FUNCTION_BLOCK FB_WatsAppResponse
VAR_INPUT
	bSend             : BOOL;
END_VAR
VAR_OUTPUT
	wind_speed		  : Lreal;
	bBusy             : BOOL;
    bError            : BOOL;
END_VAR
VAR
	fbRequest         : FB_IotHttpRequest;
    fbJson            : FB_JsonDomParser;
    nState            : UDINT;
    RisingEdge        : R_TRIG;

    bGetContentResult : BOOL;
    sContent          : STRING(511);

    bGetJsonResult    : BOOL;
    jsonDoc           : SJsonValue;
    jsonVal           : SJsonValue;
	jsonWind           : SJsonValue;

    nReqCount         : UDINT;
    nResCount         : UDINT;
    nValidResCount    : UDINT;
    nErrCount         : UDINT;
	bHasMember		  : BOOL;
	bHasMember2		  : BOOL;
END_VAR
VAR_IN_OUT
	 fbClient          : FB_IotHttpClient;
END_VAR

RisingEdge(CLK:= bSend);
CASE nState OF
0:
    IF RisingEdge.Q THEN
        IF fbRequest.SendRequest(sUri:= '/cebc385e-7c19-40b8-aaac-81ec04618ab7',
                                 fbClient:= fbClient, 
                                 eRequestType:= ETcIotHttpRequestType.HTTP_POST, 0, 0, 0) THEN
            nState:= 1;
            nReqCount:= nReqCount+1;
            bBusy:= TRUE;
            bError:= FALSE;
        END_IF
    END_IF
1:
    IF NOT fbRequest.bBusy THEN
        bError:= TRUE;
        IF NOT fbRequest.bError THEN
            bGetContentResult:= fbRequest.GetContent(pContent:= ADR(sContent), 
                                                     nContentSize:= SIZEOF(sContent), 
                                                     bSetNullTermination:= TRUE);
            IF fbRequest.nStatusCode >= 200 AND fbRequest.nStatusCode < 300 THEN
                bGetJsonResult:= FALSE;
                jsonDoc:= fbRequest.GetJsonDomContent(fbJson);
//                IF jsonDoc <> 0 THEN
//                    bHasMember := fbJson.HasMember(jsonDoc, 'current');
//					IF (bHasMember) THEN
//						bHasMember := FALSE;
//						jsonVal := fbJson.FindMember(jsonDoc, 'current');
//					END_IF
					
//					bHasMember2 := fbJson.HasMember(jsonVal, 'wind_mph');
//					IF (bHasMember2) THEN
//						bHasMember2 := FALSE;
//						jsonWind := fbJson.FindMember(jsonVal, 'wind_mph');
//						wind_speed := fbJson.GetDouble(jsonWind);
//						WindSpeed := fbJson.GetDouble(jsonWind);
//					END_IF
					
//                    nValidResCount:= nValidResCount+1;
//                    bError:= FALSE;
//                END_IF
                nResCount:= nResCount+1;
            END_IF
        END_IF
        nState:= 0;
        bBusy:= FALSE;
        IF bError THEN
            nErrCount:= nErrCount+1;
        END_IF
    END_IF
END_CASE

END_FUNCTION_BLOCK

(* stored: Version 1.1.0.1, ProductVersion 3.1.4024.12
   POU FB_WatsAppResponse: Id {7eb5ff43-6e09-43d1-ae62-39d89c0e5279}, SpecialFunc None *)
